{attribute 'strict'}
{attribute 'to_string'}
TYPE E_Kardex_Robot_Programs :
(
	NoCommand			:= 0, 	// Amíg "0"-ás a programszám addig nincs mozgási program végrehajtás, vár…
	Home				:= 1,	// Robot Zóna-6-ba megy és bemozog alaphelyzetbe
	Park				:= 2,	// Robot Zóna-6-ba megy és bemozog parkoló pozícióba.
	Service				:= 3,	// Robot elmegy szerviz pozícióba.
	KardexMeasurement	:= 4,	// Robot beméri az aktuális kardex polc koordiátáit.
	KardexPickUp 		:= 11,	// Kardex paletta kiszedés
	KardexPutDown	 	:= 12,	// Kardex paletta lerakás
	Mir_1_PickUp		:= 13,	// MIR-1 paletta kiszedés
	Mir_1_PutDown		:= 14,	// MIR-1 paletta lerakás
	Mir_2_PickUp		:= 15,	// MIR-2 paletta kiszedés
	Mir_2_PutDown		:= 16,	// MIR-2 paletta lerakás
	PufferPickUp 		:= 17,	// Puffer paletta kiszedés
	PufferPutDown		:= 18,	// Puffer paletta lerakás
	Strip_1_PickUp		:= 19,	// Szalag-1 paletta kiszedés
	Strip_1_PutDown		:= 20,	// Szalag-1 paletta lerakás
	Strip_2_PickUp		:= 21,	// Szalag-2 paletta kiszedés
	Strip_2_PutDown		:= 22,	// Szalag-2 paletta lerakás
	Strip_3_PickUp		:= 23,	// Szalag-3 paletta kiszedés
	Strip_3_PutDown		:= 24,	// Szalag-3 paletta lerakás
	Strip_3_Rotate		:= 25	// Szalag-3 paletta forgatás
);
END_TYPE

(* stored: Version 1.1.0.1, ProductVersion 3.1.4024.12
   EnumerationTextList E_Kardex_Robot_Programs: Id {32f2ff98-2c0e-4575-8e74-9fee76abe5d3} *)
